{attribute 'qualified_only'}
{attribute 'strict'}
{attribute 'to_string'}
TYPE E_OperationState :
(
	NotApplicable := 0,
	Pending,
	Processing,
	Completed,
	Failed
);
END_TYPE

(* stored: Version 1.1.0.1, ProductVersion 3.1.4026.18
   DUT E_OperationState: Id {63d676ed-4eb2-4d32-b33b-6dfc8185b576} *)
